TYPE TcaTwinSAFEStatus :
STRUCT
	Safe : BOOL;
	Error : BOOL;
	Running : BOOL;
END_STRUCT
END_TYPE

(* stored: Version 1.1.0.1
   DUT TcaTwinSAFEStatus: Id {6961313f-577e-475c-8226-09c131eeb958} *)
